// TIA Portal V19 export
TYPE "stConfigGrease"
   STRUCT
      uiNbPulsePerKm : UInt := 4411;   // Number of pulse per km
      uiKmForGreasing : UInt := 32;   // Number of Km between each greasing
      tTimeEnableGreasePump : Time := T#1M;   // Time of enabling grease pump
      tTimeoutPxGrease : Time := T#1M;   // Timeout for the proxy greas
   END_STRUCT;
END_TYPE
